Fanuc KAREL source: kb00002.KL

-- PROVISIONAL review KL for V1013-1; original PC SHA256 e6db15ab2f76e0cb3b068daf41acb146f8e5f86c5394722ad103f397f5638713
-- Incomplete behavior may be omitted. Consult companion uncertainty JSON. Do not deploy.
PROGRAM KB00002
%NOLOCKGROUP
VAR
  P1 : INTEGER
  RESULT : INTEGER
BEGIN
  -- UNRESOLVED_PC offsets 5-12; opcodes 9D,23
  -- UNRESOLVED_PC offsets 17-30; opcodes 21,50,23
  -- UNRESOLVED_PC offsets 35-39; opcodes 7F
END KB00002
